(* CoDeSys 2.3.5.6 project: lyjak_01_st.pro *)
(* Libraries: Standard.lib*31.10.14 11:17:58, SYSLIBCALLBACK.LIB*31.10.14 11:17:58 *)

(* PLC configuration (modules and I/O channels)
I1 AT %IX0.0 [LocalBitInput] Input I1
I2 AT %IX0.1 [LocalBitInput] Input I2
I3 AT %IX0.2 [LocalBitInput] Input I3
I4 AT %IX0.3 [LocalBitInput] Input I4
I5 AT %IX0.4 [LocalBitInput] Input I5
I6 AT %IX0.5 [LocalBitInput] Input I6
I7 AT %IX0.6 [LocalBitInput] Input I7
I8 AT %IX0.7 [LocalBitInput] Input I8
I9 AT %IX1.0 [LocalBitInput] Input I9
I10 AT %IX1.1 [LocalBitInput] Input I10
I11 AT %IX1.2 [LocalBitInput] Input I11
I12 AT %IX1.3 [LocalBitInput] Input I12
I13 AT %IX1.4 [LocalDiagInput] Diagnostic Input I13
I14 AT %IX1.5 [LocalDiagInput] Diagnostic Input I14
I15 AT %IX1.6 [LocalDiagInput] Diagnostic Input I15
I16 AT %IX1.7 [LocalDiagInput] Diagnostic Input I16
I7_Analog AT %IW2 [LocalAnalogIn] Input I7, 10Bit, 0-10VDC
I8_Analog AT %IW4 [LocalAnalogIn] Input I8, 10Bit, 0-10VDC
I11_Analog AT %IW6 [LocalAnalogIn] Input I11, 10Bit, 0-10VDC
I12_Analog AT %IW8 [LocalAnalogIn] Input I12, 10Bit, 0-10VDC
Transistor Outputs [EC4P_TOutputs] node 0, in %IB10 out %QB0
  Q1 AT %QX0.0 [LocalBitOutput] Transistor-Output Q1
  Q2 AT %QX0.1 [LocalBitOutput] Transistor-Output Q2
  Q3 AT %QX0.2 [LocalBitOutput] Transistor-Output Q3
  Q4 AT %QX0.3 [LocalBitOutput] Transistor-Output Q4
  Q5 AT %QX0.4 [LocalBitOutput] Transistor-Output Q5
  Q6 AT %QX0.5 [LocalBitOutput] Transistor-Output Q6
  Q7 AT %QX0.6 [LocalBitOutput] Transistor-Output Q7
  Q8 AT %QX0.7 [LocalBitOutput] Transistor-Output Q8
No Analog Output [EC4P_NoAnalogOutput] node 1, in %IB10 out %QB1
No Keys [EC4P_NoKeys] node 2, in %IB10 out %QB1
No Counter [EC4P_NoCounter] node 3, in %IB10 out %QB1
Extension [EC4P_Extension] node 1, in %IB10 out %QB1
  No Extension [EC4P_NoExtension] node 0, in %IB10 out %QB1
*)

(* POU PLC_PRG, ST *)
PROGRAM PLC_PRG
VAR
END_VAR
Q1:= I1 AND (NOT I2 OR I4) AND NOT I3;
Q2 := NOT I5 AND (I1 OR I2) AND (I2 OR I3);
Q3 := (NOT I1 OR NOT I2) AND (NOT I3 OR I4 OR I5);
Q4 := NOT I4 OR (NOT I5 AND I6);
Q5 := (I4 OR I5) AND I6 AND (I8 OR I9);
Q6 := (I4 OR I5) AND NOT I6;
Q7 := (I10 OR I11 OR I12) AND (I6 OR I5) AND (I8 OR I9 AND NOT I5);
Q8 := I1 AND (I2 OR I3) OR (I4 AND I5 OR I6 AND I3) AND (I8 AND I9 OR I10 AND I11);
END_PROGRAM
ACTION CFC:
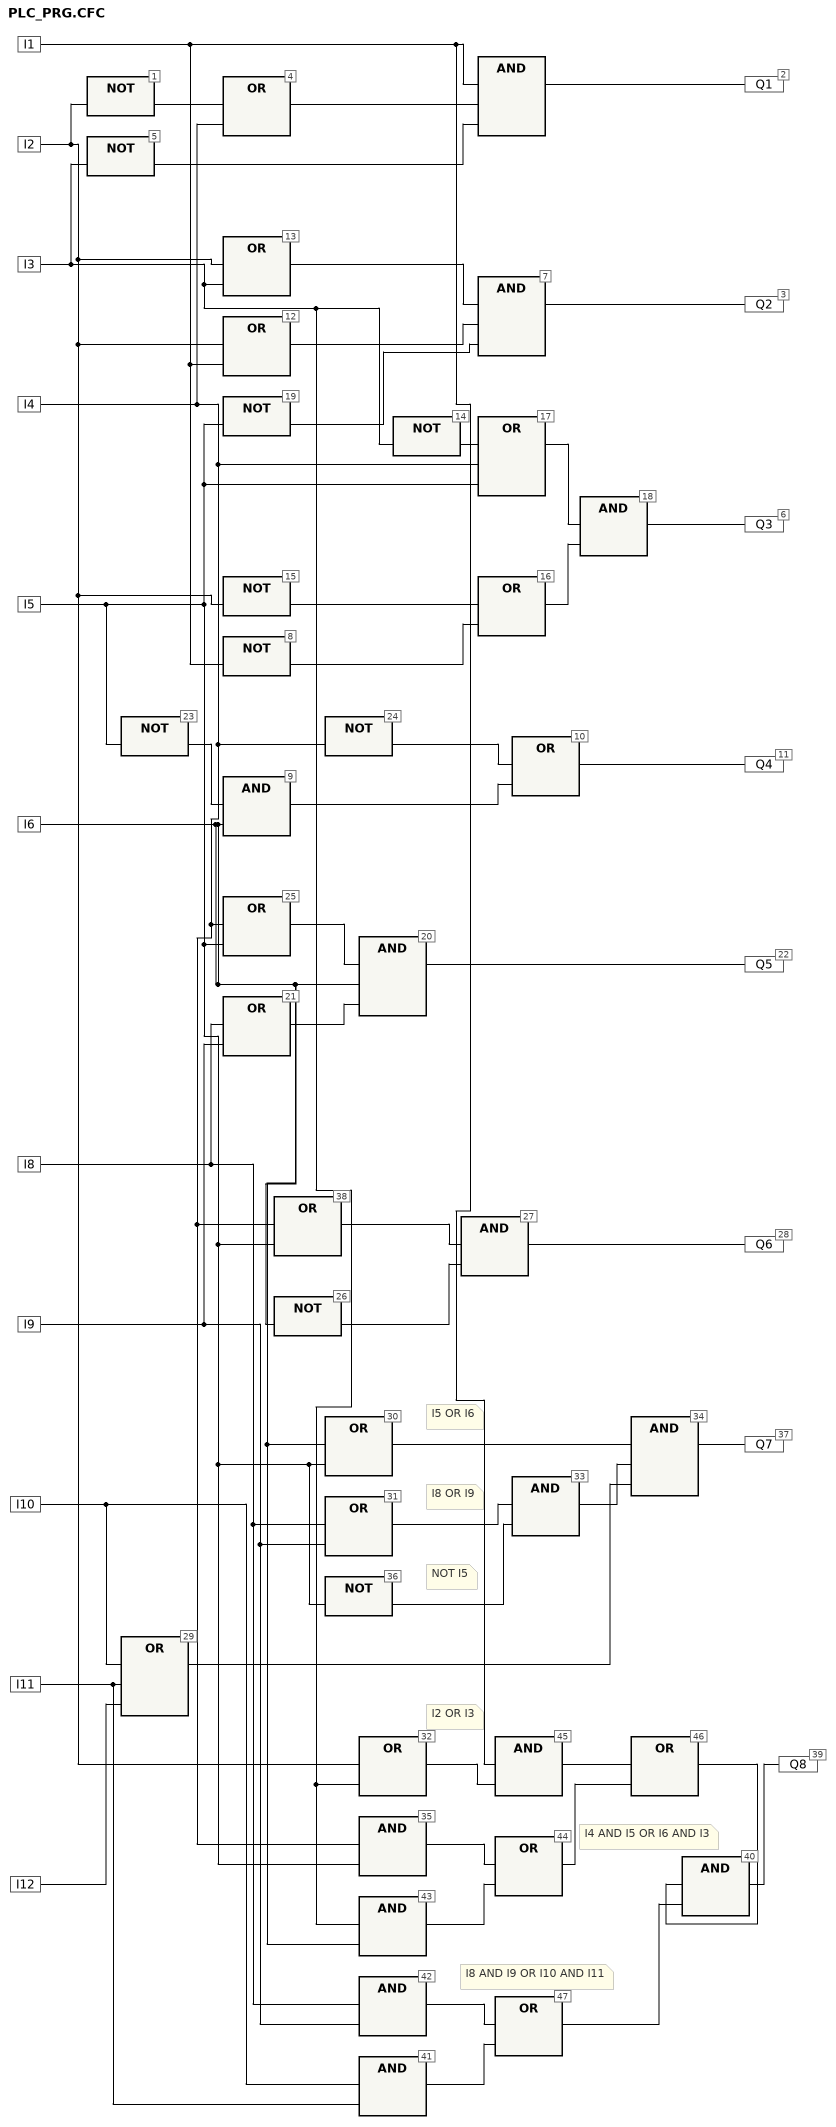
_CFC_ (* Continuous Function Chart, elements in execution order *)
(* I8 OR I9 *)
(* I5 OR I6 *)
(* NOT I5 *)
(* I2 OR I3 *)
(* I8 AND I9 OR I10 AND I11 *)
(* I4 AND I5 OR I6 AND I3 *)
#0 AND(I1, #4, #5)
#1 NOT(I2)
#2 Q1 <= #0
#3 Q2 <= #7
#4 OR(#1, I4)
#5 NOT(I3)
#6 Q3 <= #18
#7 AND(#13, #12, #19)
#8 NOT(I1)
#9 AND(#23, I6)
#10 OR(#24, #9)
#11 Q4 <= #10
#12 OR(I2, I1)
#13 OR(I2, I3)
#14 NOT(I3)
#15 NOT(I2)
#16 OR(#15, #8)
#17 OR(#14, I4, I5)
#18 AND(#17, #16)
#19 NOT(I5)
#20 AND(#25, I6, #21)
#21 OR(I8, I9)
#22 Q5 <= #20
#23 NOT(I5)
#24 NOT(I4)
#25 OR(I4, I5)
#26 NOT(I6)
#27 AND(#38, #26)
#28 Q6 <= #27
#29 OR(I10, I11, I12)
#30 OR(I6, I5)
#31 OR(I8, I9)
#32 OR(I2, I3)
#33 AND(#31, #36)
#34 AND(#30, #33, #29)
#35 AND(I4, I5)
#36 NOT(I5)
#37 Q7 <= #34
#38 OR(I4, I5)
#39 Q8 <= #40
#40 AND(#46, #47)
#41 AND(I10, I11)
#42 AND(I8, I9)
#43 AND(I3, I6)
#44 OR(#35, #43)
#45 AND(I1, #32)
#46 OR(#45, #44)
#47 OR(#42, #41)
_END_CFC_
END_ACTION
